(* CODESYS project Estação 1 - Distribution (2022).project

Project tree, tasks and I/O mapping:
  Device : CPX-CEC-C1-V3, Festo AG & Co. KG, order no. 3473128, version 3.5.7.37
      unmapped channels: Rotary switch
    application Application
      libraries: Standard, * (System)
      task MainTask (cyclic, interval t#20ms, priority 20) calls PLC_PRG
      program PLC_PRG [ST]
      global variables GVL
      function ATUALIZAR_VALORES [ST]
      program teste_comunicacao [ST]
    PLC_Diagnosis : PLC-Diagnosis, Festo AG & Co. KG, version 3.5.4.1
    CPX_System : CPX_System, Festo AG & Co. KG, order no. 3473128, version 1.258
      CEC_C1_V3 : CEC-C1-V3, Festo AG & Co. KG, order no. 3473128, version 1.258
          settings:  = 0;  = 179732921454080;  = 167946432;  = 16777215;  = 0;  = 13959208;  = 1f5477a3;  = 5
      _8DI_8DO : 8DI/8DO, Festo AG & Co. KG, order no. 526257, version 1.258
          settings:  = 0;  = 1;  = 1;  = 1;  = 1;  = 0;  = 1;  = 1;  = 0;  = 0;  = 0;  = 0;  = 0;  = 0;  = 0;  = 0;  = 0;  = 0;  = 0;  = 0;  = 0;  = 0;  = 0;  = 0;  = 0;  = 0;  = 0;  = 0;  = 0;  = 0;  = 0;  = 0;  = 0;  = 0;  = 0;  = 0;  = 0;  = 0;  = 0;  = 0;
             = 0;  = 0;  = 0;  = 0;  = 0;  = 0;  = 0;  = 0;  = 0;  = 0;  = 0;  = 0;  = 0;  = 0;  = 0;  = 0;  = 0;  = 0;  = 0;  = 0;  = 0;  = 0;  = 0;  = 0;  = 0;  = 0;  = 0;  = 0;  = 0;  = 0;  = 0;  = 0;  = 0;  = 0;  = 0;  = 0;  = 0;  = 0;  = 0;  = 0;
             = 576751027668385792;  = 'PI%i.0.0.1=1';  = 'PI%i.0.1.1=1';  = 'PI%i.0.2.1=1';  = 'PI%i.1.0.1=1';  = 'PI%i.1.1.1=0';  = 'PI%i.1.4.2=1';  = 'PI%i.1.6.2=1';  = 'PI%i.6.0.1=0';  = 'PI%i.6.1.1=0';  = 'PI%i.6.2.1=0';  = 'PI%i.6.3.1=0';  = 'PI%i.6.4.1=0';  = 'PI%i.6.5.1=0';  = 'PI%i.6.6.1=0';  = 'PI%i.6.7.1=0';  = dd30772c;  = 6
          unmapped channels: Input 0, Output 0
      _8DI_8DO_1 : 8DI/8DO, Festo AG & Co. KG, order no. 526257, version 1.258
          settings:  = 0;  = 1;  = 1;  = 1;  = 1;  = 0;  = 1;  = 1;  = 0;  = 0;  = 0;  = 0;  = 0;  = 0;  = 0;  = 0;  = 0;  = 0;  = 0;  = 0;  = 0;  = 0;  = 0;  = 0;  = 0;  = 0;  = 0;  = 0;  = 0;  = 0;  = 0;  = 0;  = 0;  = 0;  = 0;  = 0;  = 0;  = 0;  = 0;  = 0;
             = 0;  = 0;  = 0;  = 0;  = 0;  = 0;  = 0;  = 0;  = 0;  = 0;  = 0;  = 0;  = 0;  = 0;  = 0;  = 0;  = 0;  = 0;  = 0;  = 0;  = 0;  = 0;  = 0;  = 0;  = 0;  = 0;  = 0;  = 0;  = 0;  = 0;  = 0;  = 0;  = 0;  = 0;  = 0;  = 0;  = 0;  = 0;  = 0;  = 0;
             = 576751027668385792;  = 'PI%i.0.0.1=1';  = 'PI%i.0.1.1=1';  = 'PI%i.0.2.1=1';  = 'PI%i.1.0.1=1';  = 'PI%i.1.1.1=0';  = 'PI%i.1.4.2=1';  = 'PI%i.1.6.2=1';  = 'PI%i.6.0.1=0';  = 'PI%i.6.1.1=0';  = 'PI%i.6.2.1=0';  = 'PI%i.6.3.1=0';  = 'PI%i.6.4.1=0';  = 'PI%i.6.5.1=0';  = 'PI%i.6.6.1=0';  = 'PI%i.6.7.1=0';  = dd379be4;  = 6
          unmapped channels: Input 0, Output 0
    Ethernet : Ethernet, 3S - Smart Software Solutions GmbH, version 3.5.10.0
      ModbusTCP_Slave_Device : ModbusTCP Slave Device, 3S - Smart Software Solutions GmbH, version 3.5.10.0
          unmapped channels: Inputs, Outputs
*)

// Device/Application/GVL
{attribute 'qualified_only'}
VAR_GLOBAL
//Entradas
	//Sensores
	S_inicio 	AT %IX1.0 :BOOL; //Sensor de inicio da esteira
	S_meio 	 	AT %IX1.1 :BOOL; //Sensor do meio da esteira
	S_fim 		AT %IX1.2 :BOOL; //Sensor do fim da esteira
	//			AT %IX1.3 :BOOL;
	C_requado 	AT %IX1.4  :BOOL; //Cilindro requado
	C_avancado 	AT %IX1.5  :BOOL; //Cilindro avançado
	Mag_vazio  	AT %IX1.6  :BOOL; //Magazine vazio (NF)
	
	//IHM
	Start_btn 		AT	%IX2.0	:BOOL;  //Botão de start
	Stop_btn 		AT	%IX2.1	:BOOL;	//Botão de stop (NF)
	Chave 			AT	%IX2.2	:BOOL;	//Chave auto/manual
	Reset_btn 		AT	%IX2.3	:BOOL;	//Botão de reset
	I4_IHM			AT	%IX2.4	:BOOL;	//Bit de saída 4 da IHM
	I5_IHM			AT	%IX2.5	:BOOL;	//Bit de saída 5 da IHM
	I6_IHM 			AT	%IX2.6	:BOOL;	//Bit de saída 6 da IHM
	I7_IHM			AT	%IX2.7	:BOOL;	//Bit de saída 7 da IHM

//Saídas
	//Atuadorres 			
	Esteira_frente 	AT	%QX0.0	:BOOL;	//Mover a esteira para frente
	Esteira_tras 	AT	%QX0.1	:BOOL;	//Mover a esteira para tras
	Separador 	 	AT	%QX0.2	:BOOL;	//Atuar separador
	//		 		AT	%QX0.3	:BOOL;	
	Cilindro_avanca AT	%QX0.4	:BOOL;	//Avançar cilindro
	//		 		AT	%QX0.5	:BOOL;	
	//				AT	%QX0.6	:BOOL;	
	//	     		AT	%QX0.7	:BOOL;	
	
	//IHM				
	Start_LED		AT	%QX1.0	:BOOL;	//LED do botão de start
	Reset_LED 		AT	%QX1.1	:BOOL;	//LED do botão de reset
	Q1_LED 			AT	%QX1.2	:BOOL;	//LED sinalizador Q1
	Q2_LED			AT	%QX1.3	:BOOL;	//LED sinalizador Q2
	Q4_IHM			AT	%QX1.4	:BOOL;	//Saída Q4 IHM
	Q5_IHM			AT	%QX1.5	:BOOL;	//Saída Q5 IHM
	Q6_IHM			AT	%QX1.6	:BOOL;	//Saída Q6 IHM
	Q7_IHM 			AT	%QX1.7	:BOOL;	//Saída Q7 IHM
	
//MODBUS bits
	//Entradas
	Mod_I_0_0 		AT %IX4.0 : BOOL; //Start 
	Mod_I_0_1	 	AT %IX4.1 : BOOL; //Stop
	Mod_I_0_2 		AT %IX4.2 : BOOL; //Reset
	Mod_I_0_3 		AT %IX4.3 : BOOL; //Modo entrada (DESATIVADO PARA ESSA ESTAÇÃO)
	Mod_I_0_4 		AT %IX4.4 : BOOL; //Modo saída (DESATIVADO PARA ESSA ESTAÇÃO)
	Mod_I_0_5 		AT %IX4.5 : BOOL; //Teste resposta da estação - IN 
	Mod_I_0_6 		AT %IX4.6 : BOOL; 
	Mod_I_0_7 		AT %IX4.7 : BOOL;
	Mod_I_1_0 		AT %IX5.0 : BOOL;
	Mod_I_1_1 		AT %IX5.1 : BOOL;
	Mod_I_1_2 		AT %IX5.2 : BOOL;
	Mod_I_1_3 		AT %IX5.3 : BOOL;
	Mod_I_1_4 		AT %IX5.4 : BOOL;
	Mod_I_1_5	 	AT %IX5.5 : BOOL;
	Mod_I_1_6 		AT %IX5.6 : BOOL;
	Mod_I_1_7 		AT %IX5.7 : BOOL;
	
	//Saídas
	Mod_Q_0_0 		AT %QX2.0 : BOOL; //Estação iniciada 		
	Mod_Q_0_1	 	AT %QX2.1 : BOOL; // Estação parada 
	Mod_Q_0_2 		AT %QX2.2 : BOOL; //Estação em processo			
	Mod_Q_0_3 		AT %QX2.3 : BOOL; // Modo entrada (DESATIVADO PARA ESSA ESTAÇÃO)
	Mod_Q_0_4 		AT %QX2.4 : BOOL; // Modo saída (DESATIVADO PARA ESSA ESTAÇÃO)
	Mod_Q_0_5 		AT %QX2.5 : BOOL; // Teste resposta da estação - OUT
	Mod_Q_0_6 		AT %QX2.6 : BOOL; //Sesor do magazine
	Mod_Q_0_7 		AT %QX2.7 : BOOL; //Sensor do fim
	Mod_Q_1_0 		AT %QX3.0 : BOOL; 
	Mod_Q_1_1 		AT %QX3.1 : BOOL; 
	Mod_Q_1_2 		AT %QX3.2 : BOOL; 
	Mod_Q_1_3 		AT %QX3.3 : BOOL; 
	Mod_Q_1_4 		AT %QX3.4 : BOOL; 
	Mod_Q_1_5	 	AT %QX3.5 : BOOL; 
	Mod_Q_1_6 		AT %QX3.6 : BOOL; 
	Mod_Q_1_7 		AT %QX3.7 : BOOL;
	Mod_Q_2_0 		AT %QX4.0 : BOOL; 
	Mod_Q_2_1 		AT %QX4.1 : BOOL; 
	Mod_Q_2_2 		AT %QX4.2 : BOOL;
	Mod_Q_2_3 		AT %QX4.3 : BOOL; 
	Mod_Q_2_4 		AT %QX4.4 : BOOL; 
	Mod_Q_2_5	 	AT %QX4.5 : BOOL; 
	Mod_Q_2_6 		AT %QX4.6 : BOOL; //principal
	Mod_Q_2_7 		AT %QX4.7 : BOOL; //parada
	Mod_Q_3_0 		AT %QX5.0 : BOOL; //Teste de comunicação - resposta

//Variáveis de lógica
	principal: BOOL;
	parada : BOOL; 
	passo1: BOOL;	
	passo2: BOOL;
	passo3: BOOL;
	passo4: BOOL;
	passo5: BOOL;
	passo6: BOOL;
	passo7: BOOL;
	passo8: BOOL;
	
	start: BOOL; //Start geral
	stop: BOOL;  //Stop geral
	reset: BOOL; //Reset geral
	key: BOOL; //key geral

END_VAR

// Device/Application/PLC_PRG
PROGRAM PLC_PRG
VAR
	
	step1: BOOL;
	step2: BOOL;
	
	TONInst: Standard.TON;
	VarBOOL1: BOOL;
	IN: INT;
	PT: TIME;
	VarBOOL2: BOOL;
	TONInst2: TON;
	TON_2: BOOL;
	TON_1: BOOL;

	TONInst3: Ton;
	TON_3: BOOL;
	TONInst4: Ton;
	TON_4: BOOL;
END_VAR

//Programa principal da estação 1

TONInst(IN := TON_1, PT:= T#0.6S);
TONInst2(IN := TON_2, PT:= T#1.3S);
TONInst3(IN := TON_3, PT:= T#0.2S);
TONInst4(IN := TON_4, PT:= T#0.2S);


ATUALIZAR_VALORES(); //Função para atualizar os valores do MODBUS
teste_comunicacao(); //Função de teste de comunicação entre a central e essa estação


IF GVL.start  AND NOT GVL.parada AND NOT GVL.principal AND ( NOT GVL.Mag_vazio OR NOT GVL.S_fim )THEN 
	GVL.principal := TRUE; //Variável que indica que a estação está iniciada
		IF GVL.S_fim THEN //Verifica se tem alguma peça parada no fim da esteira (Sensor NF)
			GVL.passo1 := TRUE; //Começa pelo passo 1, onde a peça é colocada na esteira pelo magazine
		ELSE 
			GVL.passo6 := TRUE;//Pula para o passo responsável por dar continuidade na peça que está no fim da esteira
			TON_3 := TRUE; //Inicia o pisca pisca
		END_IF
	GVL.Q1_LED := TRUE; //Liga o LED que indica que a estação está iniciada
	GVL.Start_LED := FALSE; //Desliga o LED do botão de start
END_IF

IF  GVL.stop THEN //Caso a estação seja parada
	GVL.principal := FALSE; //Rseeta a flag que sinaliza que a estação está iniciada
	GVL.parada := TRUE; //Seta a flag de indicação de estação parada 
	GVL.Esteira_frente :=FALSE; //Para a esteira em ambos os sentidos
	GVL.Esteira_tras :=FALSE;
	GVL.Start_LED := FALSE; //Apaga o LED de start
	GVL.Reset_LED := TRUE; //Apaga o LED de reset
	GVL.Q2_LED := FALSE; //Apara o LED de indicação de processo
	GVL.Q1_LED := FALSE; //Apaga o LED de indicação de estação em processo
	TON_3 := FALSE; //Para o poisca pisca
END_IF

IF GVL.reset AND NOT GVL.principal AND GVL.parada //Reset da estação
THEN
	GVL.passo1:= FALSE; //Reseta todos os passos
	GVL.passo2:= FALSE;
	GVL.passo3:= FALSE;
	GVL.passo4:= FALSE;
	GVL.passo5:= FALSE;
	GVL.passo6:= FALSE;
	GVL.passo7:= FALSE;
	GVL.passo8:= FALSE;
	GVL.Cilindro_avanca := FALSE; //Recua o cilindro
	GVL.Separador:= FALSE; //Desliga o separador
	GVL.Esteira_frente :=FALSE; //Para as esteiras
	GVL.Esteira_tras :=FALSE;
	GVL.parada := FALSE; //Reseta a flag que sinaliza que a estação está parada

	TON_1 := FALSE;//Reseta todos os timers
	TON_2 := FALSE;
	TON_3 := FALSE;
	TON_4 := FALSE;
	GVL.Reset_LED := FALSE; //Apara o LED de reset
END_IF

IF NOT GVL.principal AND NOT GVL.parada THEN //Caso a estação esteja pronta para ser iniciada
	GVL.Start_LED := TRUE; //Liga o LED do botão de start
END_IF
	

IF GVL.principal AND NOT GVL.parada THEN  //Pisca pisca
	IF TONInst4.Q THEN
		TON_4 := FALSE;
		TON_3 := TRUE;
		GVL.Q2_LED := FALSE;
	END_IF
	IF TONInst3.Q THEN
		TON_3 := FALSE;
		TON_4 := TRUE;
		GVL.Q2_LED := TRUE;
	END_IF
END_IF


IF GVL.principal AND GVL.passo1 AND NOT GVL.parada THEN 
		GVL.passo1 := FALSE;
		GVL.passo2 := TRUE;
		GVL.Cilindro_avanca := TRUE;
		TON_3 := TRUE;
END_IF

 

IF GVL.C_avancado AND GVL.passo2 AND NOT GVL.parada THEN
		GVL.passo2 := FALSE;
		GVL.passo3 := TRUE;
		TON_1 := TRUE;
	END_IF

	IF GVL.passo3 AND TONInst.Q AND NOT GVL.parada THEN
		GVL.passo3 := FALSE;
		GVL.passo4 :=TRUE;
		GVL.Cilindro_avanca := FALSE;
		TON_1 := FALSE;
	END_IF
	
	IF GVL.C_requado AND GVL.passo4 AND NOT GVL.parada THEN
		GVL.passo4:=FALSE;
		GVL.passo5:= TRUE;
		GVL.Esteira_frente :=TRUE;
	END_IF
	
	IF NOT GVL.S_fim AND GVL.passo5 AND NOT GVL.parada THEN
		GVL.passo5 := FALSE;
		GVL.passo6 := TRUE;
		GVL.Esteira_frente :=FALSE;
	END_IF
	
	IF GVL.passo6 AND GVL.I6_IHM AND NOT GVL.parada THEN
		GVL.passo6 := FALSE;
		GVL.passo7 := TRUE;
		GVL.Esteira_frente :=TRUE;
		TON_2 := TRUE;
	END_IF
	
	IF GVL.passo7 AND TONInst2.Q AND NOT GVL.parada THEN
		TON_2 := FALSE;
		GVL.passo7 := FALSE;
		GVL.passo8 := TRUE;
		GVL.Esteira_frente :=FALSE;
	END_IF
	
	IF GVL.passo8 AND NOT GVL.Mag_vazio AND NOT GVL.parada THEN
		GVL.passo8 := FALSE;
		GVL.passo1 := TRUE;
	END_IF
	
	IF GVL.passo8 AND GVL.Mag_vazio AND NOT GVL.parada THEN
		GVL.passo8 := FALSE;
		GVL.principal := FALSE;
		GVL.Q2_LED := FALSE;
		TON_3 := FALSE;
	END_IF

END_PROGRAM

// Device/Application/ATUALIZAR_VALORES
FUNCTION ATUALIZAR_VALORES : int
VAR
END_VAR

//Ataualização de variáveis no MODBUS, indicando alguns status
GVL.Mod_Q_0_0 := GVL.principal; //Indicação de estação iniciada
GVL.Mod_Q_0_1 := GVL.parada; 	//Indicação de estação parada
GVL.Mod_Q_0_2 := GVL.principal; //Indocação de estação em processo
GVL.Mod_Q_0_6 := GVL.Mag_vazio; //Indicação de que o magazine está vazio
GVL.Mod_Q_0_7 := GVL.S_fim;		//Indicação de uma peça parada no fim da esteira do módulo 1

IF GVL.Start_btn OR GVL.Mod_I_0_0 THEN  //Atualização do valor da variável de start
	GVL.start := TRUE;
	ELSE
	GVL.start := FALSE;
END_IF

IF NOT GVL.Stop_btn OR GVL.Mod_I_0_1 THEN //Atualização do valor da variável de stop
	GVL.stop := TRUE;
	ELSE
	GVL.stop := FALSE;
END_IF

IF GVL.Reset_btn OR GVL.Mod_I_0_2 THEN //Atualização do valor da variável de reset
	GVL.reset := TRUE;
	ELSE
	GVL.reset := FALSE;	
END_IF

IF GVL.Chave OR GVL.Mod_I_0_3 THEN //Atualização do valor da variável da chave
	GVL.key := TRUE;
	ELSE
	GVL.key := FALSE;
END_IF

END_FUNCTION

// Device/Application/teste_comunicacao
PROGRAM teste_comunicacao
VAR
	
	TON_temp_1: TON;
	TON_1: BOOL;	

END_VAR

gvl.Mod_Q_0_5 := gvl.Mod_I_0_5;

END_PROGRAM
